(*
SPDX-FileCopyrightText: © 2026 Oleksandr Tiutyk <trofimich@gmail.com>
SPDX-License-Identifier: MIT
License: https://opensource.org/license/mit
*)

{attribute 'no_explicit_call' := 'do not call this function block directly'} 
FUNCTION_BLOCK IgnoreExceptionHandlingPolicy EXTENDS Object IMPLEMENTS IExceptionHandlingPolicy
VAR
	{attribute 'hide'} 
	_ClassName : STRING := __POUNAME();
END_VAR

{attribute 'monitoring' := 'call'}
PROPERTY ClassName : REFERENCE TO STRING
GET
ClassName REF= _ClassName;
END_GET
END_PROPERTY

METHOD HandleException : EXCEPTION_REACTION
VAR_INPUT
	exception : IReadOnlyException;
	handlingObject : IObject;
END_VAR
VAR_IN_OUT CONSTANT
	failedMethodName : STRING(255);
END_VAR
HandleException := EXCEPTION_REACTION.IGNORE;
END_METHOD

{attribute 'monitoring' := 'call'}
PROPERTY NamespaceName : REFERENCE TO STRING
GET
NamespaceName REF= CurrentNamespace.Name;
END_GET
END_PROPERTY

{attribute 'monitoring' := 'call'}
PROPERTY SelfSize : ULINT
GET
SelfSize := XSIZEOF(THIS^);
END_GET
END_PROPERTY

END_FUNCTION_BLOCK

(* stored: Version 1.1.0.1
   POU IgnoreExceptionHandlingPolicy: Id {73dbd0d5-9e48-4680-a175-0b9578d97a63}, SpecialFunc None
   Property ClassName: Id {43ebadc4-9a39-418f-bb26-db6ff83e7100}
   Get Get: Id {6fdc23b0-2262-49e6-b252-405331e403da}
   Method HandleException: Id {fcea6d33-f06b-4b19-b3f4-9e4986bc971d}
   Property NamespaceName: Id {37112c41-1ab9-4c45-93e4-22e01ef57382}
   Get Get: Id {12ecafbe-70a4-46e5-995e-96235a05e3ab}
   Property SelfSize: Id {af50f4b1-9365-4694-982e-ba15d20d4bb7}
   Get Get: Id {9d45ac5f-4024-473b-89b5-4d8fe61791d6} *)
